SYSTEM CONVEYORS (* System Configuration *)
  (* Standard: 61499-1 *)
  (* Version 0.4, 2009-03-05, JHC, Holobloc Inc., Deleted Application. *)
  (* Version 0.3, 2003-12-05, JHC, Rockwell Automation, Renamed from NEWSYSTEM. *)
  (* Version 0.2, 2002-11-05, JHC, Rockwell Automation, Fixed missing (empty) FBD in Application. *)
  (* Version 0.1, 2002-01-17, JHC, Rockwell Automation, Minor cleanup *)
  (* Version 0.0, 2000-05-27, JHC, Rockwell Automation *)
  DEVICE VIEW : FRAME_DEVICE(BOUNDS := [500,30,510,500], GRID := [1])
    RESOURCE VIEW_Resource : VIEW_PANEL(DIA := 50, SIZE := [10,10], VERTICAL := 0)
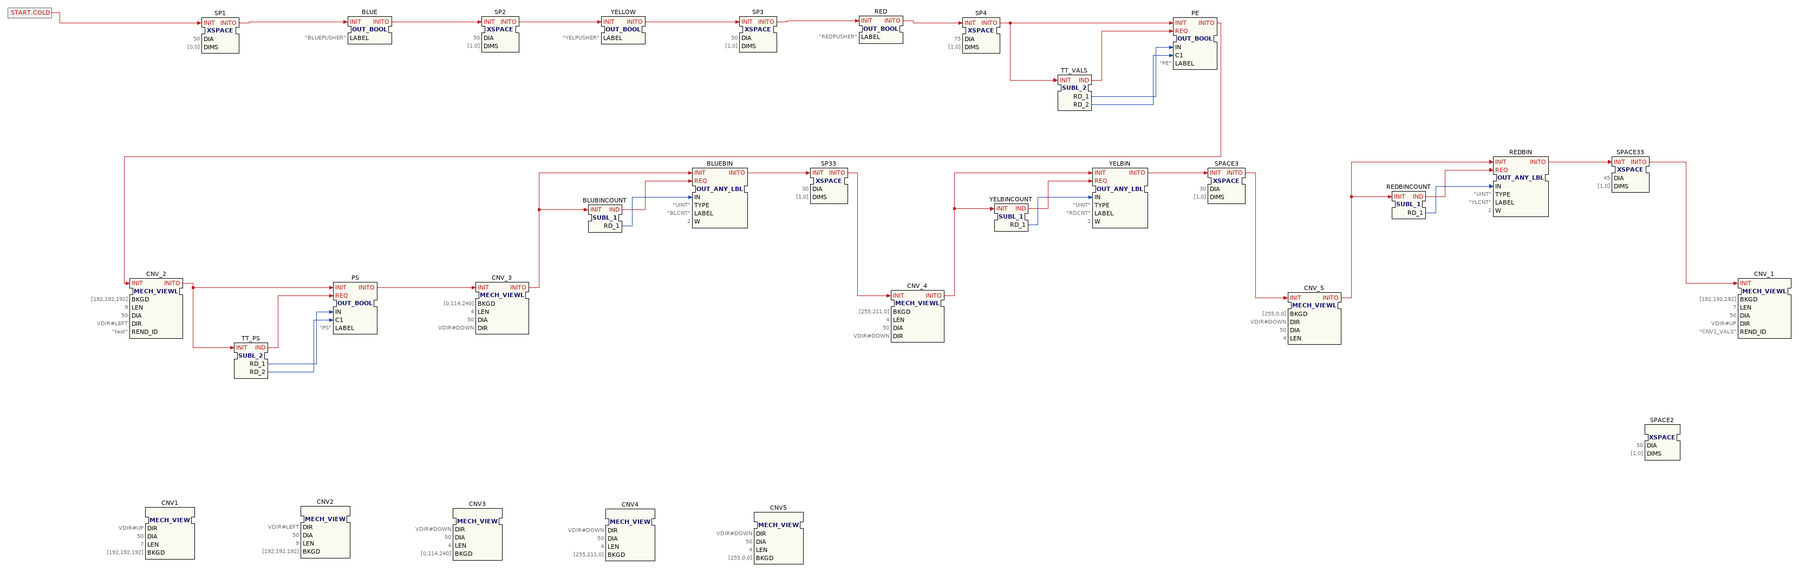
      FBS
        CNV1 : MECH_VIEW(DIR := VDIR#UP, DIA := 50, LEN := 7, BKGD := [192,192,192]);
        CNV2 : MECH_VIEW(DIR := VDIR#LEFT, DIA := 50, LEN := 9, BKGD := [192,192,192]);
        CNV3 : MECH_VIEW(DIR := VDIR#DOWN, DIA := 50, LEN := 4, BKGD := [0,114,240]);
        CNV4 : MECH_VIEW(DIR := VDIR#DOWN, DIA := 50, LEN := 4, BKGD := [255,211,0]);
        CNV5 : MECH_VIEW(DIR := VDIR#DOWN, DIA := 50, LEN := 4, BKGD := [255,0,0]);
        SPACE2 : XSPACE(DIA := 50, DIMS := [1,0]);
        SPACE3 : XSPACE(DIA := 30, DIMS := [1,0]);
        BLUE : OUT_BOOL(LABEL := "BLUEPUSHER");
        YELLOW : OUT_BOOL(LABEL := "YELPUSHER");
        RED : OUT_BOOL(LABEL := "REDPUSHER");
        SP1 : XSPACE(DIA := 50, DIMS := [0,0]);
        SP2 : XSPACE(DIA := 50, DIMS := [1,0]);
        SP3 : XSPACE(DIA := 50, DIMS := [1,0]);
        SP4 : XSPACE(DIA := 75, DIMS := [1,0]);
        SPACE33 : XSPACE(DIA := 45, DIMS := [1,0]);
        PS : OUT_BOOL(LABEL := "PS");
        PE : OUT_BOOL(LABEL := "PE");
        CNV_2 : MECH_VIEWL(BKGD := [192,192,192], LEN := 9, DIA := 50, DIR := VDIR#LEFT, REND_ID := "test");
        CNV_3 : MECH_VIEWL(BKGD := [0,114,240], LEN := 4, DIA := 50, DIR := VDIR#DOWN);
        CNV_4 : MECH_VIEWL(BKGD := [255,211,0], LEN := 4, DIA := 50, DIR := VDIR#DOWN);
        CNV_5 : MECH_VIEWL(BKGD := [255,0,0], DIR := VDIR#DOWN, DIA := 50, LEN := 4);
        CNV_1 : MECH_VIEWL(BKGD := [192,192,192], LEN := 7, DIA := 50, DIR := VDIR#UP, REND_ID := "CNV1_VALS");
        TT_VALS : SUBL_2;
        TT_PS : SUBL_2;
        YELBIN : OUT_ANY_LBL(TYPE := "UINT", LABEL := "RDCNT", W := 2);
        BLUEBIN : OUT_ANY_LBL(TYPE := "UINT", LABEL := "BLCNT", W := 2);
        SP33 : XSPACE(DIA := 30, DIMS := [1,0]);
        REDBIN : OUT_ANY_LBL(TYPE := "UINT", LABEL := "YLCNT", W := 2);
        BLUBINCOUNT : SUBL_1;
        YELBINCOUNT : SUBL_1;
        REDBINCOUNT : SUBL_1;
      END_FBS
      EVENT_CONNECTIONS
        START.COLD TO SP1.INIT;
        SP1.INITO TO BLUE.INIT;
        BLUE.INITO TO SP2.INIT;
        SP2.INITO TO YELLOW.INIT;
        YELLOW.INITO TO SP3.INIT;
        SP3.INITO TO RED.INIT;
        RED.INITO TO SP4.INIT;
        SP4.INITO TO PE.INIT;
        PE.INITO TO CNV_2.INIT;
        CNV_2.INITO TO PS.INIT;
        PS.INITO TO CNV_3.INIT;
        SPACE33.INITO TO CNV_1.INIT;
        SP4.INITO TO TT_VALS.INIT;
        TT_VALS.IND TO PE.REQ;
        CNV_2.INITO TO TT_PS.INIT;
        TT_PS.IND TO PS.REQ;
        YELBIN.INITO TO SPACE3.INIT;
        SPACE3.INITO TO CNV_5.INIT;
        CNV_4.INITO TO YELBIN.INIT;
        CNV_3.INITO TO BLUEBIN.INIT;
        BLUEBIN.INITO TO SP33.INIT;
        SP33.INITO TO CNV_4.INIT;
        CNV_5.INITO TO REDBIN.INIT;
        REDBIN.INITO TO SPACE33.INIT;
        CNV_3.INITO TO BLUBINCOUNT.INIT;
        BLUBINCOUNT.IND TO BLUEBIN.REQ;
        CNV_4.INITO TO YELBINCOUNT.INIT;
        YELBINCOUNT.IND TO YELBIN.REQ;
        REDBINCOUNT.IND TO REDBIN.REQ;
        CNV_5.INITO TO REDBINCOUNT.INIT;
      END_CONNECTIONS
      DATA_CONNECTIONS
        TT_VALS.RD_1 TO PE.IN;
        TT_VALS.RD_2 TO PE.C1;
        TT_PS.RD_1 TO PS.IN;
        TT_PS.RD_2 TO PS.C1;
        BLUBINCOUNT.RD_1 TO BLUEBIN.IN;
        YELBINCOUNT.RD_1 TO YELBIN.IN;
        REDBINCOUNT.RD_1 TO REDBIN.IN;
      END_CONNECTIONS
    END_RESOURCE
  END_DEVICE
  DEVICE HMI : FRAME_DEVICE(BOUNDS := [1010,30,600,500], GRID := [1,3])
    RESOURCE HMI_RESOURCE : VIEW_PANEL(DIA := 50, SIZE := [10,10], VERTICAL := 0)
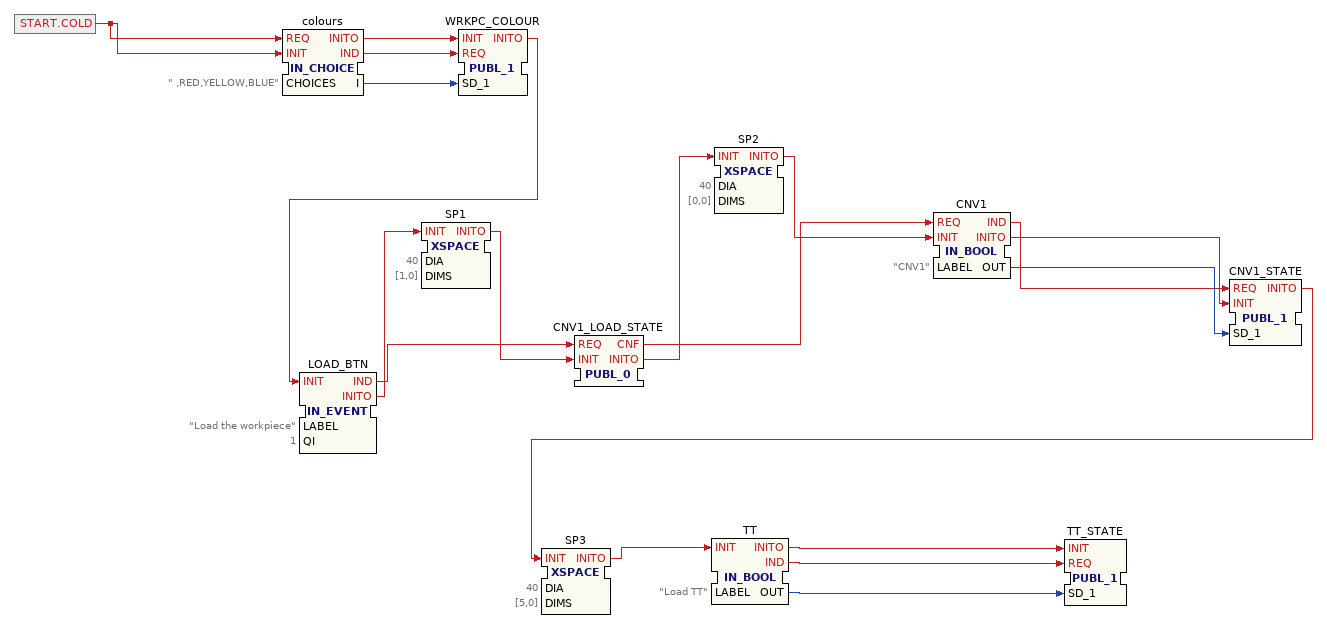
      FBS
        CNV1 : IN_BOOL(LABEL := "CNV1");
        colours : IN_CHOICE(CHOICES := " ,RED,YELLOW,BLUE");
        WRKPC_COLOUR : PUBL_1;
        LOAD_BTN : IN_EVENT(LABEL := "Load the workpiece", QI := 1);
        CNV1_STATE : PUBL_1;
        CNV1_LOAD_STATE : PUBL_0;
        TT_STATE : PUBL_1;
        TT : IN_BOOL(LABEL := "Load TT");
        SP1 : XSPACE(DIA := 40, DIMS := [1,0]);
        SP2 : XSPACE(DIA := 40, DIMS := [0,0]);
        SP3 : XSPACE(DIA := 40, DIMS := [5,0]);
      END_FBS
      EVENT_CONNECTIONS
        START.COLD TO colours.REQ;
        START.COLD TO colours.INIT;
        colours.INITO TO WRKPC_COLOUR.INIT;
        colours.IND TO WRKPC_COLOUR.REQ;
        CNV1.IND TO CNV1_STATE.REQ;
        CNV1.INITO TO CNV1_STATE.INIT;
        LOAD_BTN.IND TO CNV1_LOAD_STATE.REQ;
        CNV1_LOAD_STATE.CNF TO CNV1.REQ;
        TT.INITO TO TT_STATE.INIT;
        TT.IND TO TT_STATE.REQ;
        LOAD_BTN.INITO TO SP1.INIT;
        SP1.INITO TO CNV1_LOAD_STATE.INIT;
        WRKPC_COLOUR.INITO TO LOAD_BTN.INIT;
        CNV1_LOAD_STATE.INITO TO SP2.INIT;
        SP2.INITO TO CNV1.INIT;
        CNV1_STATE.INITO TO SP3.INIT;
        SP3.INITO TO TT.INIT;
      END_CONNECTIONS
      DATA_CONNECTIONS
        colours.I TO WRKPC_COLOUR.SD_1;
        CNV1.OUT TO CNV1_STATE.SD_1;
        TT.OUT TO TT_STATE.SD_1;
      END_CONNECTIONS
    END_RESOURCE
    RESOURCE HMI_RES : PANEL_RESOURCE(ROWS := 10, COLS := 4)
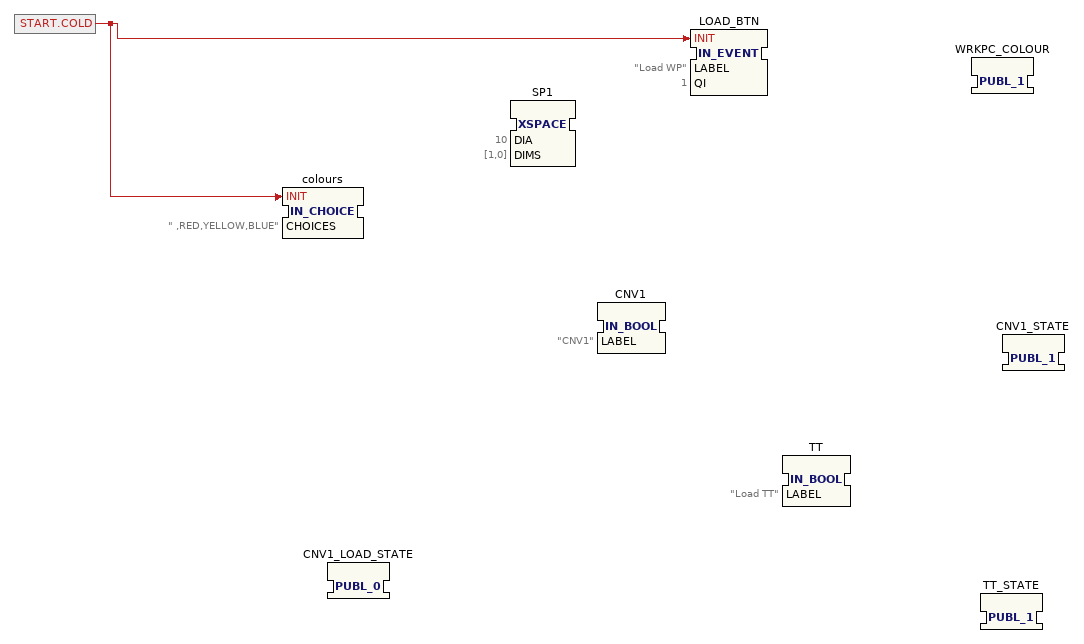
      FBS
        colours : IN_CHOICE(CHOICES := " ,RED,YELLOW,BLUE");
        WRKPC_COLOUR : PUBL_1;
        LOAD_BTN : IN_EVENT(LABEL := "Load WP", QI := 1);
        CNV1_LOAD_STATE : PUBL_0;
        CNV1 : IN_BOOL(LABEL := "CNV1");
        TT : IN_BOOL(LABEL := "Load TT");
        CNV1_STATE : PUBL_1;
        TT_STATE : PUBL_1;
        SP1 : XSPACE(DIA := 10, DIMS := [1,0]);
      END_FBS
      EVENT_CONNECTIONS
        START.COLD TO colours.INIT;
        START.COLD TO LOAD_BTN.INIT;
      END_CONNECTIONS
    END_RESOURCE
  END_DEVICE
  DEVICE MODEL : FRAME_DEVICE(BOUNDS := [500,570,500,500], GRID := [1])
    RESOURCE CONV1_MODEL : VIEW_PANEL(DIA := 50, SIZE := [1,1])
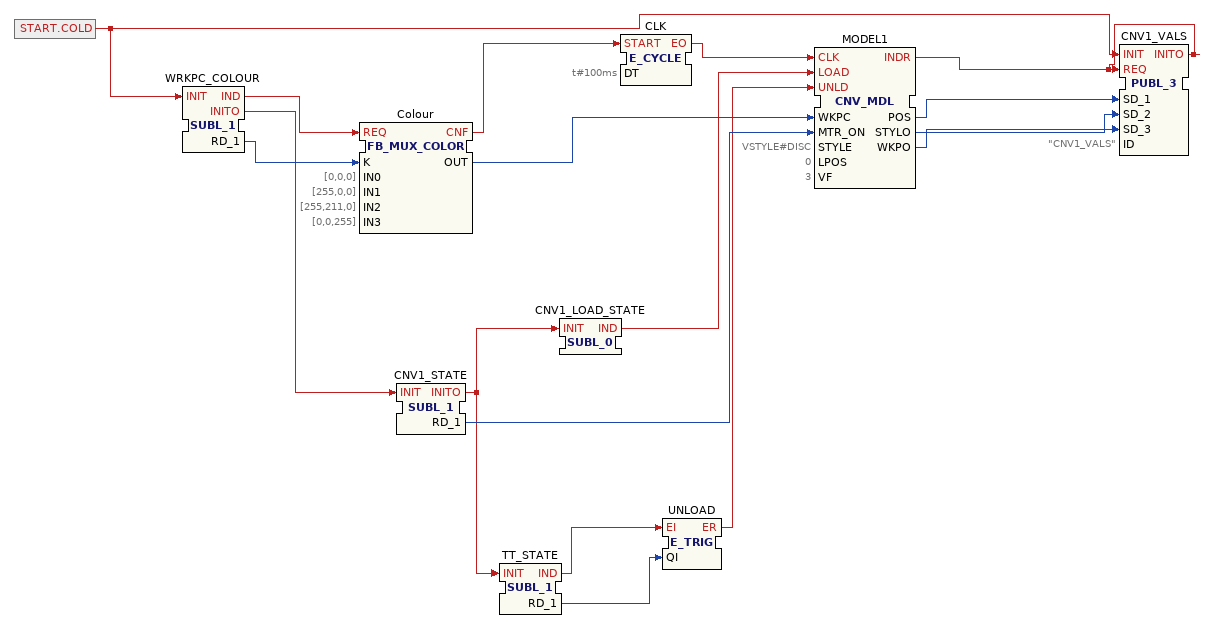
      FBS
        WRKPC_COLOUR : SUBL_1;
        Colour : FB_MUX_COLOR(IN0 := [0,0,0], IN1 := [255,0,0], IN2 := [255,211,0], IN3 := [0,0,255]);
        MODEL1 : CNV_MDL(STYLE := VSTYLE#DISC, LPOS := 0, VF := 3);
        CLK : E_CYCLE(DT := t#100ms);
        CNV1_STATE : SUBL_1;
        CNV1_LOAD_STATE : SUBL_0;
        CNV1_VALS : PUBL_3(ID := "CNV1_VALS");
        TT_STATE : SUBL_1;
        UNLOAD : E_TRIG;
      END_FBS
      EVENT_CONNECTIONS
        START.COLD TO WRKPC_COLOUR.INIT;
        WRKPC_COLOUR.IND TO Colour.REQ;
        WRKPC_COLOUR.INITO TO CNV1_STATE.INIT;
        CNV1_STATE.INITO TO CNV1_LOAD_STATE.INIT;
        Colour.CNF TO CLK.START;
        START.COLD TO CNV1_VALS.INIT;
        MODEL1.INDR TO CNV1_VALS.REQ;
        CLK.EO TO MODEL1.CLK;
        CNV1_VALS.INITO TO CNV1_VALS.REQ;
        CNV1_LOAD_STATE.IND TO MODEL1.LOAD;
        CNV1_STATE.INITO TO TT_STATE.INIT;
        TT_STATE.IND TO UNLOAD.EI;
        UNLOAD.ER TO MODEL1.UNLD;
      END_CONNECTIONS
      DATA_CONNECTIONS
        Colour.OUT TO MODEL1.WKPC;
        CNV1_STATE.RD_1 TO MODEL1.MTR_ON;
        WRKPC_COLOUR.RD_1 TO Colour.K;
        MODEL1.POS TO CNV1_VALS.SD_1;
        MODEL1.STYLO TO CNV1_VALS.SD_2;
        MODEL1.WKPO TO CNV1_VALS.SD_3;
        TT_STATE.RD_1 TO UNLOAD.QI;
      END_CONNECTIONS
    END_RESOURCE
    RESOURCE TT_MODEL : VIEW_PANEL(DIA := 50, SIZE := [1,1])
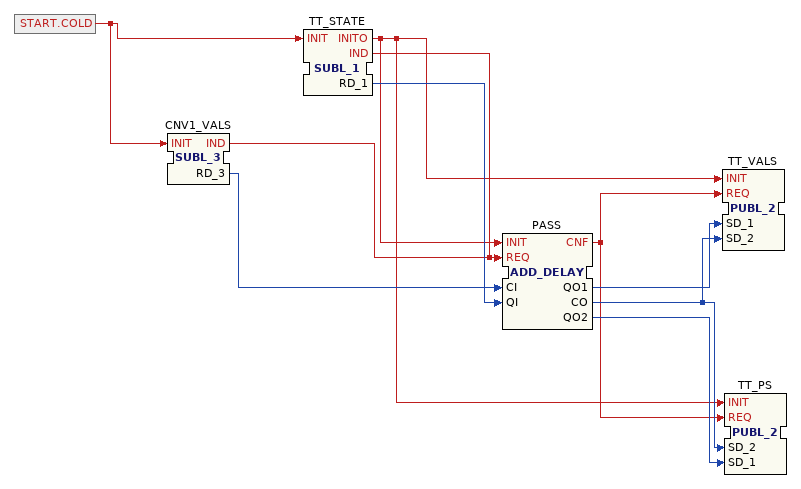
      FBS
        TT_VALS : PUBL_2;
        CNV1_VALS : SUBL_3;
        TT_STATE : SUBL_1;
        TT_PS : PUBL_2;
        PASS : ADD_DELAY;
      END_FBS
      EVENT_CONNECTIONS
        START.COLD TO CNV1_VALS.INIT;
        START.COLD TO TT_STATE.INIT;
        TT_STATE.INITO TO TT_VALS.INIT;
        TT_STATE.INITO TO TT_PS.INIT;
        TT_STATE.INITO TO PASS.INIT;
        TT_STATE.IND TO PASS.REQ;
        CNV1_VALS.IND TO PASS.REQ;
        PASS.CNF TO TT_VALS.REQ;
        PASS.CNF TO TT_PS.REQ;
      END_CONNECTIONS
      DATA_CONNECTIONS
        CNV1_VALS.RD_3 TO PASS.CI;
        TT_STATE.RD_1 TO PASS.QI;
        PASS.QO1 TO TT_VALS.SD_1;
        PASS.CO TO TT_VALS.SD_2;
        PASS.CO TO TT_PS.SD_2;
        PASS.QO2 TO TT_PS.SD_1;
      END_CONNECTIONS
    END_RESOURCE
  END_DEVICE
END_SYSTEM
